{attribute addProperty BoxType "CX5010 EtherCAT slave-1b82-0016"}
{attribute addProperty Id "TxPdoStateAT %I*BOOL8115TxPdoToggleAT %I*BOOL8116"}
{attribute addProperty CRC "2891013676"}
{attribute addProperty SizeInBites "16"}
{attribute addProperty SizeInBytes "2"}
TYPE Device_Status_Mapping_AC515E2C :
STRUCT
	{attribute addProperty Name "TxPdoState"}
	TxPdoState AT %I* : BOOL;
	{attribute addProperty Name "TxPdoToggle"}
	TxPdoToggle AT %I* : BOOL;
END_STRUCT
END_TYPE

(* stored: Version 1.2.0.0, ProductVersion 3.1.4024.9
   DUT Device_Status_Mapping_AC515E2C: Id {61b11626-e65d-4f51-9b13-e4e8bc962f1f} *)
